FUNCTION alg_a_DledQ1 : BOOL
VAR_INPUT
	state: STATE;
END_VAR

alg_a_DledQ1 := FALSE;

END_FUNCTION

(* stored: Version 1.1.0.1, ProductVersion 3.1.4022.18
   POU alg_a_DledQ1: Id {7dbf884f-666d-48b6-ad82-e480a10d9bb2}, SpecialFunc None *)
